FUNCTION_BLOCK setTimers (* Composite Function Block Type *)
  (* Standard: 61499-2 *)
  (* Version 0.2, 2003-12-05, JHC, Rockwell Automation, Renamed from NEWCOMPFB. *)
  (* Version 0.1, 2002-01-08, JHC, Rockwell Automation, Added DLY FB as example. *)
  (* Version 0.0, 2000-05-27, JHC, Rockwell Automation *)
  (* Compiler header: package fb.rt.template; *)
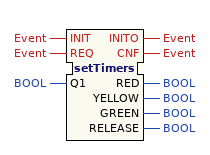
  EVENT_INPUT
    INIT; (* Initialization Request *)
    REQ; (* Normal Execution Request *)
  END_EVENT
  EVENT_OUTPUT
    INITO; (* Initialization Confirm *)
    CNF; (* Execution Confirmation *)
  END_EVENT
  VAR_INPUT
    Q1 : BOOL;
  END_VAR
  VAR_OUTPUT
    RED : BOOL;
    YELLOW : BOOL;
    GREEN : BOOL;
    RELEASE : BOOL;
  END_VAR
  FBS
    Control : TRAFFICCONTROL1;
    toGreen : E_TRIG;
    TimerGreen : E_DELAY(DT := t#3s);
    TimerYellow : E_DELAY(DT := t#1s);
  END_FBS
  EVENT_CONNECTIONS
    INIT TO Control.INIT;
    REQ TO toGreen.EI;
    toGreen.ER TO Control.T0;
    toGreen.ER TO TimerGreen.START;
    TimerGreen.EO TO Control.T1;
    TimerGreen.EO TO TimerYellow.START;
    TimerYellow.EO TO Control.T2;
    Control.INITO TO INITO;
    Control.CNF TO CNF;
  END_CONNECTIONS
  DATA_CONNECTIONS
    Control.RED TO RED;
    Control.YELLOW TO YELLOW;
    Control.GREEN TO GREEN;
    Control.Release TO RELEASE;
    Q1 TO toGreen.QI;
  END_CONNECTIONS
END_FUNCTION_BLOCK
